// TIA Portal V20 export
TYPE "LER_typeBrakeTestEmHmiCommands"
// stored: Access Published
   STRUCT
      start : Bool;
      stop : Bool;
   END_STRUCT;
END_TYPE
